# EPICS substitutions: rogueApp/Db/roguePcie.substitutions
# roguePcie.substitutions

file biDevRogue.template
{
	{
	    	NAME	= "TimingFrameRx:RxClkCount"
    		PATH	= "Top.TimingFrameRx.RxClkCount"
	    	PYPV	= "Top:TimingFrameRx:RxClkCount"
		DESC	= "Recovered clock count div 16"
	}
	{
    		NAME	= "TimingFrameRx:RxRstCount"
	    	PATH	= "Top.TimingFrameRx.RxRstCount"
	    	PYPV	= "Top:TimingFrameRx:RxRstCount"
		DESC	= "Receive link reset count"
	}
	{
		NAME	= "TrEvent:FifoOverflow"
		PATH	= "Top.TriggerEventManager.TriggerEventBuffer[0].FifoOverflow"
		PYPV	= "Top:TriggerEventManager:TriggerEventBuffer[0]:FifoOverflow"
		SCAN	= "\$(SCAN=1 second)"
	}
	{
		NAME	= "TrEvent:FifoPause"
		PATH	= "Top.TriggerEventManager.TriggerEventBuffer[0].FifoPause"
		PYPV	= "Top:TriggerEventManager:TriggerEventBuffer[0]:FifoPause"
		SCAN	= "\$(SCAN=1 second)"
	}
	{
		NAME	= "TrEvent:XpmOverflow"
		PATH	= "Top.TriggerEventManager.TriggerEventBuffer[0].XpmOverflow"
		PYPV	= "Top:TriggerEventManager:TriggerEventBuffer[0]:XpmOverflow"
		SCAN	= "\$(SCAN=1 second)"
	}
	{
		NAME	= "TrEvent:XpmPause"
		PATH	= "Top.TriggerEventManager.TriggerEventBuffer[0].XpmPause"
		PYPV	= "Top:TriggerEventManager:TriggerEventBuffer[0]:XpmPause"
		SCAN	= "\$(SCAN=1 second)"
	}
}
file boDevRogue.template
{
	{
		NAME	= "Timing:timingRxUserRst",
	    	PATH	= "Top.SystemRegs.timingRxUserRst"
    		PYPV	= "Top:SystemRegs:timingRxUserRst"
		DESC 	= "Timing RX reset"
		SAVE	= ""
	}
	{
		NAME	= "Timing:timingTxUserRst",
	    	PATH	= "Top.SystemRegs.timingTxUserRst"
	    	PYPV	= "Top:SystemRegs:timingTxUserRst"
		DESC 	= "Timing TX reset"
		SAVE	= ""
	}
	{
		NAME	= "HV:0:enable",
	    	PATH	= "Top.SystemRegs.HvEn[0]"
	    	PYPV	= "Top:SystemRegs:HvEn[0]"
		DESC 	= "HV0 enable"
		SAVE	= "VAL"
		PINI    = "YES"
	}
	{
		NAME	= "HV:1:enable",
	    	PATH	= "Top.SystemRegs.HvEn[1]"
	    	PYPV	= "Top:SystemRegs:HvEn[1]"
		DESC 	= "HV1 enable"
		SAVE	= "VAL"
		PINI    = "YES"
	}
}
file boolDevRogue.template
{
	{
		NAME	= "SystemRegs:AdcCtrl1"
		PATH	= "Top.SystemRegs.AdcCtrl1"
		PYPV	= "Top:SystemRegs:AdcCtrl1"
		ZNAM	= "False"
		ONAM	= "True"
		OSV		= "MINOR"
		DOL		= "0"
		PINI	= "YES"
		SAVE	= ""
	}
	{
		NAME	= "SystemRegs:AdcCtrl2"
		PATH	= "Top.SystemRegs.AdcCtrl2"
		PYPV	= "Top:SystemRegs:AdcCtrl2"
		ZNAM	= "False"
		ONAM	= "True"
		OSV		= "MINOR"
		DOL		= "0"
		PINI	= "YES"
		SAVE	= ""
	}
	{
		NAME	= "SystemRegs:AdcReset"
		PATH	= "Top.SystemRegs.AdcReset"
		PYPV	= "Top:SystemRegs:AdcReset"
		ZNAM	= "Normal"
		ONAM	= "Reset"
		OSV		= "MINOR"
		DOL		= "0"
		PINI	= "YES"
	}
	{
		NAME	= "SystemRegs:AvccEn0"
		PATH	= "Top.SystemRegs.AvccEn0"
		PYPV	= "Top:SystemRegs:AvccEn0"
		DESC	= "Enable AVCC0 DCDC"
		ZSV		= "MINOR"
		DOL		= "1"
		PINI	= "YES"
	}
	{
		NAME	= "SystemRegs:AvccEn1"
		PATH	= "Top.SystemRegs.AvccEn1"
		PYPV	= "Top:SystemRegs:AvccEn1"
		DESC	= "Enable AVCC1 DCDC"
		ZSV		= "MINOR"
		DOL		= "1"
		PINI	= "YES"
	}
	{
		NAME	= "SystemRegs:Ap5V5En"
		PATH	= "Top.SystemRegs.Ap5V5En"
		PYPV	= "Top:SystemRegs:Ap5V5En"
		DESC	= "Enable analog buffers 5.5V DCDC"
		ZSV		= "MINOR"
		DOL		= "1"
		PINI	= "YES"
	}
	{
		NAME	= "SystemRegs:Ap5V0En"
		PATH	= "Top.SystemRegs.Ap5V0En"
		PYPV	= "Top:SystemRegs:Ap5V0En"
		DESC	= "Enable analog buffers 5.0V LDO"
		ZSV		= "MINOR"
		DOL		= "1"
		PINI	= "YES"
	}
	{
		NAME	= "SystemRegs:A0p3V3En"
		PATH	= "Top.SystemRegs.A0p3V3En"
		PYPV	= "Top:SystemRegs:A0p3V3En"
		DESC	= "Enable ADCs analog 3.3V LDO"
		ZSV		= "MINOR"
		DOL		= "1"
		PINI	= "YES"
	}
	{
		NAME	= "SystemRegs:A1p3V3En"
		PATH	= "Top.SystemRegs.A1p3V3En"
		PYPV	= "Top:SystemRegs:A1p3V3En"
		DESC	= "Enable ADCs analog 3.3V LDO"
		ZSV		= "MINOR"
		DOL		= "1"
		PINI	= "YES"
	}
	{
		NAME	= "SystemRegs:Ap1V8En"
		PATH	= "Top.SystemRegs.Ap1V8En"
		PYPV	= "Top:SystemRegs:Ap1V8En"
		DESC	= "Enable ADCs analog 1.8V LDO"
		ZSV		= "MINOR"
		DOL		= "1"
		PINI	= "YES"
	}
	{
		NAME	= "SystemRegs:FpgaTmpCritLatch"
		PATH	= "Top.SystemRegs.FpgaTmpCritLatch"
		PYPV	= "Top:SystemRegs:FpgaTmpCritLatch"
		DESC	= "FPGA Critical Temperature Triggered"
	}
	{
		NAME	= "Timing:UseMiniTpg",
		PATH	= "Top.SystemRegs.timingUseMiniTpg"
		PYPV	= "Top:SystemRegs:timingUseMiniTpg"
		PINI	= "YES"
		SAVE	= "VAL"
		SCAN	= ""
	}
	{
		NAME	= "TrEvent:MasterEnable"
		PATH	= "Top.TriggerEventManager.TriggerEventBuffer[0].MasterEnable"
		PYPV	= "Top:TriggerEventManager:TriggerEventBuffer[0]:MasterEnable"
		DOL 	= "1"
		PINI	= "YES"
		SAVE	= "VAL"
		SCAN	= ""
	}
	{
		NAME	= "SystemRegs:TrigEn",
		PATH	= "Top.SystemRegs.TrigEn"
		PYPV	= "Top:SystemRegs:TrigEn"
		DOL 	= "1"
		PINI	= "YES"
		SAVE	= "VAL"
		SCAN	= ""
	}
	{
		NAME	= "EvrV2:EnableTrig",
		PATH	= "Top.TriggerEventManager.EvrV2CoreTriggers.EvrV2TriggerReg[0].EnableTrig"
		PYPV	= "Top:TriggerEventManager:EvrV2CoreTriggers:EvrV2TriggerReg[0]:EnableTrig"
		DESC	= "Enables the EvrV2 Trigger Output"
		DOL		= "1"
		PINI	= "YES"
		SAVE	= ""
		SCAN	= "\$(SCAN=1 second)"
	}
	{
		NAME	= "RawBuffers:BuffEn0",
		PATH	= "Top.RawBuffers.BuffEn[0]"
		PYPV	= "Top:RawBuffers:BuffEn[0]"
		DOL 	= "1"
		PINI	= "YES"
		SAVE	= "VAL"
		SCAN	= ""
	}
	{
		NAME	= "RawBuffers:BuffEn1",
		PATH	= "Top.RawBuffers.BuffEn[1]"
		PYPV	= "Top:RawBuffers:BuffEn[1]"
		DOL 	= "1"
		PINI	= "YES"
		SAVE	= "VAL"
		SCAN	= ""
	}
	{
		NAME	= "RawBuffers:BuffEn2",
		PATH	= "Top.RawBuffers.BuffEn[2]"
		PYPV	= "Top:RawBuffers:BuffEn[2]"
		DOL 	= "1"
		PINI	= "YES"
		SAVE	= "VAL"
		SCAN	= ""
	}
	{
		NAME	= "RawBuffers:BuffEn3",
		PATH	= "Top.RawBuffers.BuffEn[3]"
		PYPV	= "Top:RawBuffers:BuffEn[3]"
		DOL 	= "1"
		PINI	= "YES"
		SAVE	= "VAL"
		SCAN	= ""
	}
	{
		NAME	= "RawBuffers:BuffEn4",
		PATH	= "Top.RawBuffers.BuffEn[4]"
		PYPV	= "Top:RawBuffers:BuffEn[4]"
		DOL 	= "1"
		PINI	= "YES"
		SAVE	= "VAL"
		SCAN	= ""
	}
	{
		NAME	= "RawBuffers:BuffEn5",
		PATH	= "Top.RawBuffers.BuffEn[5]"
		PYPV	= "Top:RawBuffers:BuffEn[5]"
		DOL 	= "1"
		PINI	= "YES"
		SAVE	= "VAL"
		SCAN	= ""
	}
	{
		NAME	= "RawBuffers:BuffEn6",
		PATH	= "Top.RawBuffers.BuffEn[6]"
		PYPV	= "Top:RawBuffers:BuffEn[6]"
		DOL 	= "1"
		PINI	= "YES"
		SAVE	= "VAL"
		SCAN	= ""
	}
	{
		NAME	= "RawBuffers:BuffEn7",
		PATH	= "Top.RawBuffers.BuffEn[7]"
		PYPV	= "Top:RawBuffers:BuffEn[7]"
		DOL 	= "1"
		PINI	= "YES"
		SAVE	= "VAL"
		SCAN	= ""
	}
	{
		NAME	= "RawBuffers:CntRst",
		PATH	= "Top.RawBuffers.CntRst"
		PYPV	= "Top:RawBuffers:CntRst"
		SCAN	= "\$(SCAN=1 second)"
	}
	{
		NAME	= "XpmMini:HwEnable",
		PATH	= "Top.XpmMiniWrapper.XpmMini.HwEnable"
		PYPV	= "Top:XpmMiniWrapper:XpmMini:HwEnable"
		PINI	= "YES"
	}
	{
		NAME	= "XpmMini:Config_L0Select_Enabled",
		PATH	= "Top.XpmMiniWrapper.XpmMini.Config_L0Select_Enabled"
		PYPV	= "Top:XpmMiniWrapper:XpmMini:Config_L0Select_Enabled"
		PINI	= "YES"
	}
}

# TODO: Move PgpRx:FrameCnt to int64DevRogue.template
file liDevRogue.template
{
	{
		NAME	= "RawBuffers:FifoPauseCnt",
		PATH	= "Top.RawBuffers.FifoPauseCnt"
		PYPV	= "Top:RawBuffers:FifoPauseCnt"
		SCAN	= "\$(SCAN=1 second)"
	}
	{
		NAME	= "SystemRegs:TempAnaRaw0",
		PATH	= "Top.SystemRegs.TempAnaRaw[0]"
		PYPV	= "Top:SystemRegs:TempAnaRaw[0]"
		DESC	= "Analog board temperature sensor 0"
		SCAN	= "\$(SCAN=1 second)"
	}
	{
		NAME	= "SystemRegs:TempAnaRaw1",
		PATH	= "Top.SystemRegs.TempAnaRaw[1]"
		PYPV	= "Top:SystemRegs:TempAnaRaw[1]"
		DESC	= "Analog board temperature sensor 1"
		SCAN	= "\$(SCAN=1 second)"
	}
	{
		NAME	= "SystemRegs:TempDigRaw0",
		PATH	= "Top.SystemRegs.TempDigRaw[0]"
		PYPV	= "Top:SystemRegs:TempDigRaw[0]"
		DESC	= "Digital board temperature sensor 0"
		SCAN	= "\$(SCAN=1 second)"
	}
	{
		NAME	= "SystemRegs:TempDigRaw1",
		PATH	= "Top.SystemRegs.TempDigRaw[1]"
		PYPV	= "Top:SystemRegs:TempDigRaw[1]"
		DESC	= "Digital board temperature sensor 1"
		SCAN	= "\$(SCAN=1 second)"
	}
	{
		NAME	= "Timing:RxLinkUp",
		PATH	= "Top.TimingFrameRx.RxLinkUp"
		PYPV	= "Top:TimingFrameRx:RxLinkUp"
		DESC	= "Timing fiber link status"
		SCAN	= "\$(SCAN=1 second)"
		LLSV 	= "MAJOR"
	}
	{
		NAME	= "TrEvent:FifoWrCnt"
		PATH	= "Top.TriggerEventManager.TriggerEventBuffer[0].FifoWrCnt"
		PYPV	= "Top:TriggerEventManager:TriggerEventBuffer[0]:FifoWrCnt"
		SCAN	= "\$(SCAN=1 second)"
	}
	{
		NAME	= "TrEvent:L0Count"
		PATH	= "Top.TriggerEventManager.TriggerEventBuffer[0].L0Count"
		PYPV	= "Top:TriggerEventManager:TriggerEventBuffer[0]:L0Count"
		SCAN	= "\$(SCAN=1 second)"
	}
	{
		NAME	= "TrEvent:L1AcceptCount"
		PATH	= "Top.TriggerEventManager.TriggerEventBuffer[0].L1AcceptCount"
		PYPV	= "Top:TriggerEventManager:TriggerEventBuffer[0]:L1AcceptCount"
		SCAN	= "\$(SCAN=1 second)"
	}
	{
		NAME	= "TrEvent:L1RejectCount"
		PATH	= "Top.TriggerEventManager.TriggerEventBuffer[0].L1RejectCount"
		PYPV	= "Top:TriggerEventManager:TriggerEventBuffer[0]:L1RejectCount"
		SCAN	= "\$(SCAN=1 second)"
	}
	{
		NAME	= "TrEvent:NotPauseToTrig"
		PATH	= "Top.TriggerEventManager.TriggerEventBuffer[0].NotPauseToTrig"
		PYPV	= "Top:TriggerEventManager:TriggerEventBuffer[0]:NotPauseToTrig"
		SCAN	= "\$(SCAN=1 second)"
	}
	{
		NAME	= "TrEvent:PauseToTrig"
		PATH	= "Top.TriggerEventManager.TriggerEventBuffer[0].PauseToTrig"
		PYPV	= "Top:TriggerEventManager:TriggerEventBuffer[0]:PauseToTrig"
		SCAN	= "\$(SCAN=1 second)"
	}
	{
		NAME	= "TrEvent:XpmMsg:PartitionDelay0"
		PATH	= "Top.TriggerEventManager.XpmMessageAligner.PartitionDelay[0]"
		PYPV	= "Top:TriggerEventManager:XpmMessageAligner:PartitionDelay[0]"
		SCAN	= "\$(SCAN=1 second)"
	}
	{
		NAME	= "TrEvent:XpmMsg:PartitionDelay1"
		PATH	= "Top.TriggerEventManager.XpmMessageAligner.PartitionDelay[1]"
		PYPV	= "Top:TriggerEventManager:XpmMessageAligner:PartitionDelay[1]"
		SCAN	= "\$(SCAN=1 second)"
	}
	{
		NAME	= "TrEvent:XpmMsg:PartitionDelay2"
		PATH	= "Top.TriggerEventManager.XpmMessageAligner.PartitionDelay[2]"
		PYPV	= "Top:TriggerEventManager:XpmMessageAligner:PartitionDelay[2]"
		SCAN	= "\$(SCAN=1 second)"
	}
	{
		NAME	= "TrEvent:XpmMsg:PartitionDelay3"
		PATH	= "Top.TriggerEventManager.XpmMessageAligner.PartitionDelay[3]"
		PYPV	= "Top:TriggerEventManager:XpmMessageAligner:PartitionDelay[3]"
		SCAN	= "\$(SCAN=1 second)"
	}
	{
		NAME	= "TrEvent:XpmMsg:PartitionDelay4"
		PATH	= "Top.TriggerEventManager.XpmMessageAligner.PartitionDelay[4]"
		PYPV	= "Top:TriggerEventManager:XpmMessageAligner:PartitionDelay[4]"
		SCAN	= "\$(SCAN=1 second)"
	}
	{
		NAME	= "TrEvent:XpmMsg:PartitionDelay5"
		PATH	= "Top.TriggerEventManager.XpmMessageAligner.PartitionDelay[5]"
		PYPV	= "Top:TriggerEventManager:XpmMessageAligner:PartitionDelay[5]"
		SCAN	= "\$(SCAN=1 second)"
	}
	{
		NAME	= "TrEvent:XpmMsg:PartitionDelay6"
		PATH	= "Top.TriggerEventManager.XpmMessageAligner.PartitionDelay[6]"
		PYPV	= "Top:TriggerEventManager:XpmMessageAligner:PartitionDelay[6]"
		SCAN	= "\$(SCAN=1 second)"
	}
	{
		NAME	= "TrEvent:XpmMsg:PartitionDelay7"
		PATH	= "Top.TriggerEventManager.XpmMessageAligner.PartitionDelay[7]"
		PYPV	= "Top:TriggerEventManager:XpmMessageAligner:PartitionDelay[7]"
		SCAN	= "\$(SCAN=1 second)"
	}
}

file loDevRogue.template
{
	{
		NAME	= "Timing:C_RxReset",
		PATH	= "Top.TimingFrameRx.C_RxReset"
		PYPV	= "Top:TimingFrameRx:C_RxReset"
		SAVE	= ""
	}
	{
		NAME	= "TrEvent:FifoReset"
		PATH	= "Top.TriggerEventManager.TriggerEventBuffer[0].FifoReset"
		PYPV	= "Top:TriggerEventManager:TriggerEventBuffer[0]:FifoReset"
		SAVE	= ""
	}
	{
		NAME	= "TrEvent:ResetCounters"
		PATH	= "Top.TriggerEventManager.TriggerEventBuffer[0].ResetCounters"
		PYPV	= "Top:TriggerEventManager:TriggerEventBuffer[0]:ResetCounters"
		SAVE	= ""
	}
}

file longDevRogue.template
{
	{
		NAME	= "EvrV2:Polarity",
		PATH	= "Top.TriggerEventManager.EvrV2CoreTriggers.EvrV2TriggerReg[0].Polarity"
		PYPV	= "Top:TriggerEventManager:EvrV2CoreTriggers:EvrV2TriggerReg[0]:Polarity"
		DESC	= "Trigger Polarity"
		SAVE	= "VAL"
		SCAN	= "\$(SCAN=1 second)"
	}
	{
		NAME	= "EvrV2:Source",
		PATH	= "Top.TriggerEventManager.EvrV2CoreTriggers.EvrV2TriggerReg[0].Source"
		PYPV	= "Top:TriggerEventManager:EvrV2CoreTriggers:EvrV2TriggerReg[0]:Source"
		DESC	= "Trigger Source"
		DOL	= "0"
		SAVE	= "VAL"
		SCAN	= "\$(SCAN=1 second)"
	}
	{
		NAME	= "RawBuffers:OvflCntBuff0",
		PATH	= "Top.RawBuffers.OvflCntBuff[0]"
		PYPV	= "Top:RawBuffers:OvflCntBuff[0]"
		SAVE	= ""
		SCAN	= "\$(SCAN=1 second)"
	}
	{
		NAME	= "RawBuffers:OvflCntBuff1",
		PATH	= "Top.RawBuffers.OvflCntBuff[1]"
		PYPV	= "Top:RawBuffers:OvflCntBuff[1]"
		SAVE	= ""
		SCAN	= "\$(SCAN=1 second)"
	}
	{
		NAME	= "RawBuffers:OvflCntBuff2",
		PATH	= "Top.RawBuffers.OvflCntBuff[2]"
		PYPV	= "Top:RawBuffers:OvflCntBuff[2]"
		SAVE	= ""
		SCAN	= "\$(SCAN=1 second)"
	}
	{
		NAME	= "RawBuffers:OvflCntBuff3",
		PATH	= "Top.RawBuffers.OvflCntBuff[3]"
		PYPV	= "Top:RawBuffers:OvflCntBuff[3]"
		SAVE	= ""
		SCAN	= "\$(SCAN=1 second)"
	}
	{
		NAME	= "RawBuffers:OvflCntBuff4",
		PATH	= "Top.RawBuffers.OvflCntBuff[4]"
		PYPV	= "Top:RawBuffers:OvflCntBuff[4]"
		SAVE	= ""
		SCAN	= "\$(SCAN=1 second)"
	}
	{
		NAME	= "RawBuffers:OvflCntBuff5",
		PATH	= "Top.RawBuffers.OvflCntBuff[5]"
		PYPV	= "Top:RawBuffers:OvflCntBuff[5]"
		SAVE	= ""
		SCAN	= "\$(SCAN=1 second)"
	}
	{
		NAME	= "RawBuffers:OvflCntBuff6",
		PATH	= "Top.RawBuffers.OvflCntBuff[6]"
		PYPV	= "Top:RawBuffers:OvflCntBuff[6]"
		SAVE	= ""
		SCAN	= "\$(SCAN=1 second)"
	}
	{
		NAME	= "RawBuffers:OvflCntBuff7",
		PATH	= "Top.RawBuffers.OvflCntBuff[7]"
		PYPV	= "Top:RawBuffers:OvflCntBuff[7]"
		SAVE	= ""
		SCAN	= "\$(SCAN=1 second)"
	}
	{
		NAME	= "RawBuffers:BuffLen",
		PATH	= "Top.RawBuffers.BuffLen"
		PYPV	= "Top:RawBuffers:BuffLen"
		DOL	= "255"
		SAVE	= "VAL"
		SCAN	= "\$(SCAN=1 second)"
	}
	{
		NAME	= "RawBuffers:FifoPauseThreshold",
		PATH	= "Top.RawBuffers.FifoPauseThreshold"
		PYPV	= "Top:RawBuffers:FifoPauseThreshold"
		PINI	= "YES"
		DOL	= "255"
		SAVE	= "VAL"
		SCAN	= ""
	}
	{
		NAME	= "RawBuffers:TrigPrescale",
		PATH	= "Top.RawBuffers.TrigPrescale"
		PYPV	= "Top:RawBuffers:TrigPrescale"
		SAVE	= "VAL"
		SCAN	= ""
	}
	{
		NAME	= "SystemRegs:TrigDelay",
		PATH	= "Top.SystemRegs.TrigDelay"
		PYPV	= "Top:SystemRegs:TrigDelay"
		PINI	= "YES"
		SAVE	= "VAL"
		SCAN	= ""
		SCAN	= "\$(SCAN=1 second)"
	}
	{
		NAME	= "Timing:RxDown",
		PATH	= "$(PTOP).TimingFrameRx.RxDown"
		PYPV	= "$(PTOP):TimingFrameRx:RxDown"
		DESC	= "Timing fiber link status"
		SCAN	= "\$(SCAN=1 second)"
		SAVE	= ""
	}
	{
		NAME	= "Timing:RxPllReset",
		PATH	= "$(PTOP).TimingFrameRx.RxPllReset"
		PYPV	= "$(PTOP):TimingFrameRx:RxPllReset"
		SCAN	= "\$(SCAN=1 second)"
		SAVE	= ""
	}
	{
		NAME	= "TrEvent:Partition"
		PATH	= "Top.TriggerEventManager.TriggerEventBuffer[0].Partition"
		PYPV	= "Top:TriggerEventManager:TriggerEventBuffer[0]:Partition"
		SAVE	= "VAL"
		SCAN	= ""
	}
	{
		NAME	= "TrEvent:PauseThreshold"
		PATH	= "Top.TriggerEventManager.TriggerEventBuffer[0].PauseThreshold"
		PYPV	= "Top:TriggerEventManager:TriggerEventBuffer[0]:PauseThreshold"
		SAVE	= "VAL"
		SCAN	= ""
	}
	{
		NAME	= "XpmMini:Config_L0Select_DestSel",
		DOL		= "32768"
		PATH	= "Top.XpmMiniWrapper.XpmMini.Config_L0Select_DestSel"
		PYPV	= "Top:XpmMiniWrapper:XpmMini:Config_L0Select_DestSel"
	}
	{
		NAME	= "XpmMini:Link",
		PATH	= "Top.XpmMiniWrapper.XpmMini.Link"
		PYPV	= "Top:XpmMiniWrapper:XpmMini:Link"
	}
	{
		NAME    = "DataPathCtrl:EnableStream"
		PATH    = "Top.DataPathCtrl.EnableStream"
		PYPV    = "Top:DataPathCtrl:EnableStream"
		SAVE    = "VAL"
		PINI    = "YES"
		SDIS    = "$(P)$(R)AxiVersion:FpgaVersion_GE_204"
		DISV    = "0"
		DRVH    = "3"
		HOPR    = "3"
	}
}

file int64InDevRogue.template
{
	{
		NAME	= "RawBuffers:TrigCnt",
		PATH	= "Top.RawBuffers.TrigCnt"
		PYPV	= "Top:RawBuffers:TrigCnt"
		SCAN	= "\$(SCAN=1 second)"
	}
	{
		NAME	= "EvrV2:Count",
		PATH	= "Top.TriggerEventManager.EvrV2CoreChannels.EvrV2ChannelReg[0].Count"
		PYPV	= "Top:TriggerEventManager:EvrV2CoreChannels:EvrV2ChannelReg[0]:Count"
		DESC	= "Count for Start of Timing Frame"
		SCAN	= "\$(SCAN=1 second)"
	}
	{
		NAME	= "Timing:sofCount",
		PATH	= "Top.TimingFrameRx.sofCount"
		PYPV	= "Top:TimingFrameRx:sofCount"
		DESC	= "Count for Start of Timing Frame"
		SCAN	= "\$(SCAN=1 second)"
	}
	{
		NAME	= "Timing:eofCount",
		PATH	= "Top.TimingFrameRx.eofCount"
		PYPV	= "Top:TimingFrameRx:eofCount"
		DESC	= "Count for End of Timing Frame"
		SCAN	= "\$(SCAN=1 second)"
	}
	{
		NAME	= "Timing:FidCount",
		PATH	= "Top.TimingFrameRx.FidCount"
		PYPV	= "Top:TimingFrameRx:FidCount"
		DESC	= "Fiducial Count"
		SCAN	= "\$(SCAN=1 second)"
	}
	{
		NAME	= "TrEvent:TriggerCount"
		PATH	= "Top.TriggerEventManager.TriggerEventBuffer[0].TriggerCount"
		PYPV	= "Top:TriggerEventManager:TriggerEventBuffer[0]:TriggerCount"
		SCAN	= "\$(SCAN=1 second)"
	}
	{
		NAME	= "TrEvent:TransitionCount"
		PATH	= "Top.TriggerEventManager.TriggerEventBuffer[0].TransitionCount"
		PYPV	= "Top:TriggerEventManager:TriggerEventBuffer[0]:TransitionCount"
		SCAN	= "\$(SCAN=1 second)"
	}
	{
		NAME	= "TrEvent:XpmMessageCount"
		PATH	= "Top.TriggerEventManager.TriggerEventBuffer[0].XpmMessageCount"
		PYPV	= "Top:TriggerEventManager:TriggerEventBuffer[0]:XpmMessageCount"
		SCAN	= "\$(SCAN=1 second)"
	}
	{
		NAME	= "TrEvent:XpmMsg:RxId"
		PATH	= "Top.TriggerEventManager.XpmMessageAligner.RxId"
		PYPV	= "Top:TriggerEventManager:XpmMessageAligner:RxId"
		SCAN	= "\$(SCAN=1 second)"
	}
}
file int64DevRogue.template
{
	{
		NAME	= "TrEvent:XpmMsg:TxId"
		PATH	= "Top.TriggerEventManager.XpmMessageAligner.TxId"
		PYPV	= "Top:TriggerEventManager:XpmMessageAligner:TxId"
		SCAN	= "\$(SCAN=1 second)"
		SAVE	= ""
	}
}

file calcin.template
{
	{
		CNAME	= "HV:0:Feedback"
		NAME	= "HV:0:FeedbackRaw"
		PATH	= "Top.HV[0].HvFeedbackRaw"
		PYPV	= "Top:HV[0]:HvFeedbackRaw"
		SCAN	= "\$(SCAN=1 second)"
		CALC    = "500.0*A/65535"
		EGU     = "V"
		SDIS    = "$(P)$(R)HV:0:enable"
		DISV    = "0"
        }
	{
		CNAME	= "HV:1:Feedback"
		NAME	= "HV:1:FeedbackRaw"
		PATH	= "Top.HV[1].HvFeedbackRaw"
		PYPV	= "Top:HV[1]:HvFeedbackRaw"
		SCAN	= "\$(SCAN=1 second)"
		CALC    = "500.0*A/65535"
		EGU     = "V"
		SDIS    = "$(P)$(R)HV:1:enable"
		DISV    = "0"
        }
}

file calcout.template
{
	{
		CNAME	= "HV:0:Control"
		NAME	= "HV:0:ControlRaw"
		PATH	= "Top.HV[0].HvControlRaw"
		PYPV	= "Top:HV[0]:HvControlRaw"
		SCAN	= ""
		CSAVE   = "VAL DRVH HOPR"
		EGU     = "V"
		CALC    = "4095*A/500.0"
		SDIS    = "$(P)$(R)HV:0:enable"
		DISV    = "0"
		DRVH    = "100"
		HOPR    = "100"
        }
	{
		CNAME	= "HV:1:Control"
		NAME	= "HV:1:ControlRaw"
		PATH	= "Top.HV[1].HvControlRaw"
		PYPV	= "Top:HV[1]:HvControlRaw"
		SCAN	= ""
		CSAVE   = "VAL DRVH HOPR"
		EGU     = "V"
		CALC    = "4095*A/500.0"
		SDIS    = "$(P)$(R)HV:1:enable"
		DISV    = "0"
		DRVH    = "100"
		HOPR    = "100"
        }
}
file longcalc.template
{
        {
                CNAME   = "TrEvent:TriggerDelayControl"
                NAME    = "TrEvent:TriggerDelay",
                PATH    = "Top.TriggerEventManager.TriggerEventBuffer[0].TriggerDelay"
                PYPV    = "Top:TriggerEventManager:TriggerEventBuffer[0]:TriggerDelay"
                DESC    = "Trigger Delay"
                SAVE    = "VAL"
                SCAN    = "\$(SCAN=1 second)"
                CSAVE   = "VAL"
                EGU     = "ns"
                CALC    = "A*1.3/7"
		LCNAME	= "TrEvent:TriggerDelayControlReadback"
		LCALC	= "A*7/1.3"
		PREC	= "4"
        }
}
#       DESC    = "0         1         2         3         "
#       DESC    = "01234567890123 Max 40 char 7890123456789"
